FUNCTION TryConvert_DT_TO_STRING : BOOL
VAR_INPUT
	in : DT;
	out : REFERENCE TO STRING;
END_VAR

out := DT_TO_STRING(in);
TryConvert_DT_TO_STRING := TRUE;

END_FUNCTION

(* stored: Version 1.1.0.1, ProductVersion 3.1.4024.12
   POU TryConvert_DT_TO_STRING: Id {8a6df26a-245b-44c3-8c72-0861336b15a3}, SpecialFunc None *)
